KUKA KRL data list: Station20.dat

&ACCESS RV
DEFDAT  Station20 PUBLIC

ENDDAT
